// TIA Portal V20 export
ORGANIZATION_BLOCK "Startup"   // OB1010, LAD, Startup
TITLE = "Complete Restart"
AUTHOR : ERsystem_FA2_DH. Kim
// stored: AutoNumber false, IsIECCheckEnabled true, Namespace Unit1.Em1, SetENOAutomatically false
   VAR_INPUT
      LostRetentive : Bool;   // True if retentive data are lost
      LostRTC : Bool;   // True if date and time are lost
   END_VAR
BEGIN

REGION Network 1 (SCL): Build the Absolut Reference Designator
   // Set the Absoult Reference Designator in the Config DB
   IF LEN(IN := "Unit1.Em1.Config".em.referenceDesignator.parent) <> 0 THEN
     "Unit1.Em1.Config".em.referenceDesignator.combined := CONCAT_WSTRING(IN1 := "Unit1.Em1.Config".em.referenceDesignator.parent, IN2 := WSTRING#'.', IN3 := "Unit1.Em1.Config".em.referenceDesignator.relative);
   ELSE
     "Unit1.Em1.Config".em.referenceDesignator.combined := "Unit1.Em1.Config".em.referenceDesignator.relative;
   END_IF;
END_REGION

REGION Network 2 (SCL): Assign axes data
   //Assign axes
   "Unit1.Em1.Config".axis[1] := "BA040AZSDR2_UnwinderBottomAxisB";

   // Assign configuration data of axis
   // 
   // Axis 1 BA030A_UnwinderVirtual
   // 
   // Axis 2 BA030AZSDR2_UnwinderBottomAxisB
   "Unit1.Em1.HmiInterface".cmUnwinderBtmAxisB.commandConfiguration.jog.velocity := 10.0;
   "Unit1.Em1.HmiInterface".cmUnwinderBtmAxisB.commandConfiguration.jog.acceleration := 100.0;
   "Unit1.Em1.HmiInterface".cmUnwinderBtmAxisB.commandConfiguration.jog.deceleration := 100.0;
   "Unit1.Em1.HmiInterface".cmUnwinderBtmAxisB.commandConfiguration.moveVelocity.velocity := 10.0;
   "Unit1.Em1.HmiInterface".cmUnwinderBtmAxisB.commandConfiguration.moveVelocity.acceleration := 100.0;
   "Unit1.Em1.HmiInterface".cmUnwinderBtmAxisB.commandConfiguration.moveVelocity.deceleration := 100.0;
   "Unit1.Em1.HmiInterface".cmUnwinderBtmAxisB.commandConfiguration.posRelative.velocity := 10.0;
   "Unit1.Em1.HmiInterface".cmUnwinderBtmAxisB.commandConfiguration.posRelative.acceleration := 100.0;
   "Unit1.Em1.HmiInterface".cmUnwinderBtmAxisB.commandConfiguration.posRelative.deceleration := 100.0;

   // FB Enable
   "Unit1.Em1.HmiInterface".cmUnwinderBtmAxisB.commands.enableMasterControl := TRUE;
END_REGION

REGION Network 3 (SCL): Assign TwoWayActuator data
   //Assgin Configuration data of TwoWayActuator
   "Unit1.Em1.Config".cmAirShaftBtmOnOff.disableFeedbackHomePos := TRUE;
   "Unit1.Em1.Config".cmAirShaftBtmOnOff.disableFeedbackWorkPos := TRUE;
END_REGION

REGION Network 4 (SCL): Assign EPC Config
   "Unit1.Em1.Config".cmEpcBtm.hwID.EkrOut_Auto_Sp_Acp_HW_ID := 1058;
   "Unit1.Em1.Config".cmEpcBtm.hwID.EkrOut_CAM_Data_HW_ID := 1059;
   "Unit1.Em1.Config".cmEpcBtm.hwID.EkrOut_CLS_Data_HW_ID := 1060;
   "Unit1.Em1.Config".cmEpcBtm.hwID.EkrOut_Guiding_edges_HW_ID := 1062;
   "Unit1.Em1.Config".cmEpcBtm.hwID.EkrOut_HEADER_Data_HW_ID := 1063;
   "Unit1.Em1.Config".cmEpcBtm.hwID.EkrOut_POS_unit_HW_ID := 1065;
   "Unit1.Em1.Config".cmEpcBtm.hwID.EkrOut_SEN_Data_HW_ID := 1066;
   "Unit1.Em1.Config".cmEpcBtm.hwID.EkrOut_Servo_Center_HW_ID := 1067;
   "Unit1.Em1.Config".cmEpcBtm.hwID.EkrOut_Setpoint_HW_ID := 1068;
   "Unit1.Em1.Config".cmEpcBtm.hwID.EkrOut_Web_width_HW_ID := 1069;
   "Unit1.Em1.Config".cmEpcBtm.hwID.EkrIn_Auto_Sp_Acp_HW_ID := 1070;
   "Unit1.Em1.Config".cmEpcBtm.hwID.EkrIn_HEADER_Data_HW_ID := 1072;
   "Unit1.Em1.Config".cmEpcBtm.hwID.EkrIn_POS_unit_HW_ID := 1074;
   "Unit1.Em1.Config".cmEpcBtm.hwID.EkrIn_Setpoint_HW_ID := 1075;
   "Unit1.Em1.Config".cmEpcBtm.hwID.EkrIn_Web_width_HW_ID := 1076;
END_REGION
END_ORGANIZATION_BLOCK
